FUNCTION F_Voltage : REAL
VAR_INPUT
	V_Reading				: INT;
END_VAR
VAR
END_VAR

// Calvin - F_Voltage
// Rev 1.0 - April 6, 2023

F_Voltage					:= INT_TO_REAL(V_Reading) / 65.534;

END_FUNCTION

(* stored: Version 1.1.0.1, ProductVersion 3.1.4024.12
   POU F_Voltage: Id {aad6c2b5-4cfe-40fe-83b6-60455098db85}, SpecialFunc None *)
